// TIA Portal project "Multi_PLC_OPC_UA_Project" (V17)

(* hardware
DEVICE "S7-1200 station_1"  S7-1200 Station
   slot 0: "Rack_0"  S7-1200 Rack  Rack  V1.0
   slot 1: "PLC1_Loading"  CPU 1214C DC/DC/DC  6ES7 214-1AG40-0XB0  V4.5
DEVICE "S7-1200 station_2"  S7-1200 Station
   slot 0: "Rack_0"  S7-1200 Rack  Rack  V1.0
   slot 1: "PLC2_Testing"  CPU 1214C DC/DC/DC  6ES7 214-1AG40-0XB0  V4.5
DEVICE "HMI_Main"  KTP700 Basic PN
   slot 0: "HMI_Main"  KTP700 Basic PN  6AV2 123-2GB03-0AX0  17.0.0.0
   slot 1: "HMI_RT_1"  KTP700 Basic PN  6AV2 123-2GB03-0AX0  17.0.0.0
   slot 5: "HMI_Main.IE_CP_1"  PROFINET Interface  17.0.0.0
      slot 1: "PROFINET Interface_1"  PROFINET Interface
         slot 1: "Port_1"  Port
*)

// ===== PLC "PLC1_Loading"  CPU 1214C DC/DC/DC =====

VAR_GLOBAL   // PLC tag table "Default tag table"
   "PB_Start_Physical" AT %I0.0 : Bool;
   "PB_Stop_Physical" AT %I0.1 : Bool;
   "Conveyor_Run" AT %Q0.0 : Bool;
   "Light_Green" AT %Q0.1 : Bool;
   "Part_Sensor" AT %I0.2 : Bool;
   "Clock_Byte" AT %MB10 : Byte;
   "Clock_10Hz" AT %M10.0 : Bool;
   "Clock_5Hz" AT %M10.1 : Bool;
   "Clock_2.5Hz" AT %M10.2 : Bool;
   "Clock_2Hz" AT %M10.3 : Bool;
   "Clock_1.25Hz" AT %M10.4 : Bool;
   "Clock_1Hz" AT %M10.5 : Bool;
   "Clock_0.625Hz" AT %M10.6 : Bool;
   "Clock_0.5Hz" AT %M10.7 : Bool;
END_VAR

DATA_BLOCK "DB_PLC1_Commands"   // DB1
{ S7_Optimized_Access := 'FALSE' }
VERSION : 0.1
   VAR
      PB_Start : Bool;
      PB_Stop : Bool;
   END_VAR
BEGIN
END_DATA_BLOCK

DATA_BLOCK "DB_PLC1_Status"   // DB2
{ S7_Optimized_Access := 'FALSE' }
VERSION : 0.1
   VAR
      Conveyor_Run : Bool;
      Part_Sensor : Bool;
      Light_Green : Bool;
      Machine_Status : Int;
   END_VAR
BEGIN
END_DATA_BLOCK

DATA_BLOCK "DB_PLC1_To_PLC2"   // DB3
{ S7_Optimized_Access := 'FALSE' }
VERSION : 0.1
   VAR
      Part_Ready : Bool;
   END_VAR
BEGIN
END_DATA_BLOCK

DATA_BLOCK "DB_From_PLC2"   // DB6
{ S7_Optimized_Access := 'FALSE' }
VERSION : 0.1
   VAR
      Part_Done : Bool;
   END_VAR
BEGIN
END_DATA_BLOCK

ORGANIZATION_BLOCK "Main"   // OB1, LAD, ProgramCycle
TITLE = "Main Program Sweep (Cycle)"
{ S7_Optimized_Access := 'TRUE' }
VERSION : 0.1
   VAR_INPUT
      Initial_Call : Bool;   // Initial call of this OB
      Remanence : Bool;   // =True, if remanent data are available
   END_VAR
BEGIN

REGION Network 1
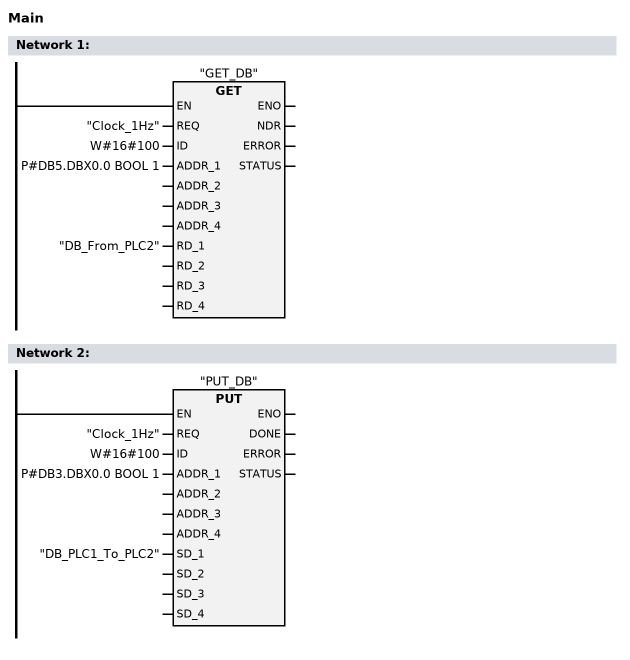
   "GET_DB"(REQ := "Clock_1Hz", ID := W#16#100, ADDR_1 := P#DB5.DBX0.0 BOOL 1, RD_1 := "DB_From_PLC2");   // GET
END_REGION

REGION Network 2
   "PUT_DB"(REQ := "Clock_1Hz", ID := W#16#100, ADDR_1 := P#DB3.DBX0.0 BOOL 1, SD_1 := "DB_PLC1_To_PLC2");   // PUT
END_REGION

REGION Network 3 (SCL)
   "DB_PLC1_Commands".PB_Start := "PB_Start_Physical";
   "DB_PLC1_Commands".PB_Stop := "PB_Stop_Physical";

   "Part_Sensor" := "DB_PLC1_Status".Part_Sensor;

   IF "DB_PLC1_Commands".PB_Start THEN

       "DB_PLC1_Status".Conveyor_Run := TRUE;
       "DB_PLC1_Status".Light_Green := TRUE;
       "DB_PLC1_Status".Machine_Status := 1;

   END_IF;

   IF "DB_PLC1_Commands".PB_Stop THEN

       "DB_PLC1_Status".Conveyor_Run := FALSE;
       "DB_PLC1_Status".Light_Green := FALSE;

       "DB_PLC1_To_PLC2".Part_Ready := FALSE;

       "DB_PLC1_Status".Machine_Status := 0;

   END_IF;


   IF "DB_PLC1_Status".Part_Sensor  AND NOT "DB_PLC1_To_PLC2".Part_Ready THEN

       "DB_PLC1_Status".Conveyor_Run := FALSE;

       "DB_PLC1_To_PLC2".Part_Ready := TRUE;

   END_IF;

   IF "DB_PLC1_To_PLC2".Part_Ready THEN

       "DB_PLC1_Status".Conveyor_Run := FALSE;

   END_IF;


   IF "DB_From_PLC2".Part_Done THEN


       "DB_PLC1_To_PLC2".Part_Ready := FALSE;

   END_IF;


   IF NOT "DB_PLC1_To_PLC2".Part_Ready
       AND "DB_PLC1_Commands".PB_Start THEN

       "DB_PLC1_Status".Conveyor_Run := TRUE;

   END_IF;


   "Conveyor_Run" := "DB_PLC1_Status".Conveyor_Run;

   "Light_Green" := "DB_PLC1_Status".Light_Green;
END_REGION
END_ORGANIZATION_BLOCK

// ===== PLC "PLC2_Testing"  CPU 1214C DC/DC/DC =====

VAR_GLOBAL   // PLC tag table "Default tag table"
   "PB_Start_Physical" AT %I0.0 : Bool;
   "PB_Stop_Physical" AT %I0.1 : Bool;
   "Conveyor_Run" AT %Q0.0 : Bool;
   "Light_Red" AT %Q0.1 : Bool;
   "Clock_Byte" AT %MB10 : Byte;
   "Clock_10Hz" AT %M10.0 : Bool;
   "Clock_5Hz" AT %M10.1 : Bool;
   "Clock_2.5Hz" AT %M10.2 : Bool;
   "Clock_2Hz" AT %M10.3 : Bool;
   "Clock_1.25Hz" AT %M10.4 : Bool;
   "Clock_1Hz" AT %M10.5 : Bool;
   "Clock_0.625Hz" AT %M10.6 : Bool;
   "Clock_0.5Hz" AT %M10.7 : Bool;
END_VAR

DATA_BLOCK "DB_PLC2_Commands"   // DB1
{ S7_Optimized_Access := 'FALSE' }
VERSION : 0.1
   VAR
      PB_Start : Bool;
      PB_Stop : Bool;
   END_VAR
BEGIN
END_DATA_BLOCK

DATA_BLOCK "DB_PLC2_Status"   // DB2
{ S7_Optimized_Access := 'FALSE' }
VERSION : 0.1
   VAR
      Conveyor_Run : Bool;
      Part_Ready_Old : Bool;
      Light_Red : Bool;
      Part_Count_Tested : Int;
      Quality_Pass : Bool;
      Machine_Status : Int;
   END_VAR
BEGIN
END_DATA_BLOCK

DATA_BLOCK "DB_From_PLC1"   // DB3
{ S7_Optimized_Access := 'FALSE' }
VERSION : 0.1
   VAR
      Part_Ready : Bool;
   END_VAR
BEGIN
END_DATA_BLOCK

DATA_BLOCK "DB_PLC2_To_PLC1"   // DB5
{ S7_Optimized_Access := 'FALSE' }
VERSION : 0.1
   VAR
      Part_Done : Bool;
   END_VAR
BEGIN
END_DATA_BLOCK

DATA_BLOCK "testing_sequence_DB"   // DB7
{ S7_Optimized_Access := 'TRUE' }
VERSION : 0.1
// stored: InstanceOfName testing_sequence
"testing_sequence"
BEGIN
END_DATA_BLOCK

FUNCTION_BLOCK "testing_sequence"   // FB1, SCL
{ S7_Optimized_Access := 'TRUE' }
VERSION : 0.1
   VAR
      "Step" : Int;
      Process_Timer : TON_TIME;
   END_VAR
BEGIN
   "DB_PLC2_Commands".PB_Start := "PB_Start_Physical";
   "DB_PLC2_Commands".PB_Stop := "PB_Stop_Physical";


   IF "DB_PLC2_Commands".PB_Start THEN

       "DB_PLC2_Status".Conveyor_Run := TRUE;
       "DB_PLC2_Status".Light_Red := TRUE;
       "DB_PLC2_Status".Machine_Status := 1;

   END_IF;


   IF "DB_PLC2_Commands".PB_Stop THEN

       "DB_PLC2_Status".Conveyor_Run := FALSE;
       "DB_PLC2_Status".Light_Red := FALSE;
       "DB_PLC2_Status".Machine_Status := 0;

       #Step := 0;

       #Process_Timer(
                      IN := FALSE,
                      PT := T#2s
       );

       "DB_PLC2_To_PLC1".Part_Done := FALSE;

   END_IF;


   CASE #Step OF

       0:
           #Process_Timer(
                          IN := FALSE,
                          PT := T#2s
           );

           "DB_PLC2_To_PLC1".Part_Done := FALSE;


           IF "DB_From_PLC1".Part_Ready THEN
               "DB_PLC2_Status".Part_Count_Tested :=
               "DB_PLC2_Status".Part_Count_Tested + 1;

               #Step := 10;

           END_IF;

       10:

           #Process_Timer(
                          IN := TRUE,
                          PT := T#2s
           );

           IF #Process_Timer.Q THEN
               #Step := 20;

           END_IF;

       20:
           #Process_Timer(
                          IN := FALSE,
                          PT := T#2s
           );

           "DB_PLC2_To_PLC1".Part_Done := TRUE;

           #Step := 30;

       30:
           IF NOT "DB_From_PLC1".Part_Ready THEN

               "DB_PLC2_To_PLC1".Part_Done := FALSE;

               #Step := 0;

           END_IF;

       ELSE

           #Step := 0;

           #Process_Timer(
                          IN := FALSE,
                          PT := T#2s
           );

           "DB_PLC2_To_PLC1".Part_Done := FALSE;

   END_CASE;
END_FUNCTION_BLOCK

ORGANIZATION_BLOCK "Main"   // OB1, LAD, ProgramCycle
TITLE = "Main Program Sweep (Cycle)"
{ S7_Optimized_Access := 'TRUE' }
VERSION : 0.1
   VAR_INPUT
      Initial_Call : Bool;   // Initial call of this OB
      Remanence : Bool;   // =True, if remanent data are available
   END_VAR
BEGIN

REGION Network 1
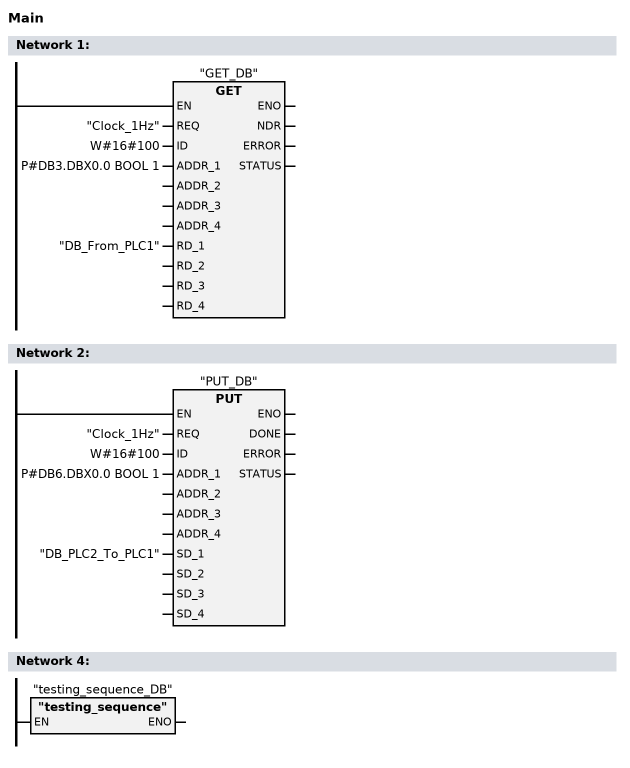
   "GET_DB"(REQ := "Clock_1Hz", ID := W#16#100, ADDR_1 := P#DB3.DBX0.0 BOOL 1, RD_1 := "DB_From_PLC1");   // GET
END_REGION

REGION Network 2
   "PUT_DB"(REQ := "Clock_1Hz", ID := W#16#100, ADDR_1 := P#DB6.DBX0.0 BOOL 1, SD_1 := "DB_PLC2_To_PLC1");   // PUT
END_REGION

REGION Network 3 (SCL)
   IF "GET_DB".ERROR THEN
       "DB_PLC2_Status".Machine_Status := 2;
   END_IF;
END_REGION

REGION Network 4
   RUNG wire#powerrail
      "testing_sequence_DB"()
   END_RUNG
   // the same network as SCL:
   "testing_sequence_DB"();   // "testing_sequence"
END_REGION
END_ORGANIZATION_BLOCK

(* ===== HMI "HMI_RT_1" =====
system functions are stored by id; their names below are inferred from use
connection "HMI_Connection_1": ETHERNET, SMART_S7_1200_OMS
connection "HMI_Connection_2": ETHERNET, SMART_S7_1200_OMS

HMI tags "Default tag table"
   "Tag_ScreenNumber" : UInt, internal
   "DB_PLC1_Commands_PB_Start" : Bool = PLC DB_PLC1_Commands.PB_Start AT %DB1.DBX0.0, 1 s
   "DB_PLC1_Commands_PB_Stop" : Bool = PLC DB_PLC1_Commands.PB_Stop AT %DB1.DBX0.1, 1 s
   "DB_PLC1_Status_Part_Count" : Int = PLC DB_PLC1_Status.Part_Count AT %DB2.DBW2, 1 s
   "DB_PLC2_Commands_PB_Start" : Bool = PLC DB_PLC2_Commands.PB_Start AT %DB1.DBX0.0, 1 s
   "DB_PLC2_Commands_PB_Stop" : Bool = PLC DB_PLC2_Commands.PB_Stop AT %DB1.DBX0.1, 1 s
   "DB_PLC2_Status_Part_Count_Tested" : Int = PLC DB_PLC2_Status.Part_Count_Tested AT %DB2.DBW2, 1 s
   "DB_From_PLC2_Part_Done" : Bool = PLC DB_From_PLC2.Part_Done AT %DB6.DBX0.0, 1 s
   "DB_PLC1_To_PLC2_Part_Ready" : Bool = PLC DB_PLC1_To_PLC2.Part_Ready AT %DB3.DBX0.0, 1 s
   "DB_PLC1_Status_Part_Count_not_tested" : Int = PLC DB_PLC1_Status.Part_Count AT %DB2.DBW2, 1 s
   "DB_PLC1_Status_Part_Sensor" : Bool = PLC DB_PLC1_Status.Part_Sensor AT %DB2.DBX0.1, 1 s
   "DB_PLC1_Status_Conveyor_Run" : Bool = PLC DB_PLC1_Status.Conveyor_Run AT %DB2.DBX0.0, 1 s
   "DB_PLC2_Status_Conveyor_Run" : Bool = PLC DB_PLC2_Status.Conveyor_Run AT %DB2.DBX0.0, 1 s
   "DB_From_PLC1_Part_Ready" : Bool = PLC DB_From_PLC1.Part_Ready AT %DB3.DBX0.0, 1 s

Template "Template_1" 800x480
   Button "Exit" at 714,429 size 71x50; TextOff 'Exit'; PictureOff "ExitRuntime_KTP700_Basic_PN_TR"; PictureOn "ExitRuntime_KTP700_Basic_PN_TR"
      on Release: StopRuntime(0)
   Button "Template_Button" at 614,429 size 71x50; TextOff 'Text'
   Button "Template_Button_1" at 514,429 size 71x50; TextOff 'Text'
   Button "Template_Button_2" at 414,429 size 71x50; TextOff 'Text'
   Button "Template_Button_3" at 314,429 size 71x50; TextOff 'Text'
   Button "Template_Button_4" at 214,429 size 71x50; TextOff 'Text'
   Button "Alarms" at 114,429 size 71x50; TextOff 'Alarms'; PictureOff "AlarmDisplay_KTP700_Basic_PN_TR"; PictureOn "AlarmDisplay_KTP700_Basic_PN_TR"
      on Release: function_ef3f5d25("Alarm window_Unacknowledged", -1)
   Button "Start screen" at 14,429 size 71x50; TextOff 'Start screen'; PictureOff "NavigateHome_KTP700_Basic_PN_TR"; PictureOn "NavigateHome_KTP700_Basic_PN_TR"
      on Release: ActivateScreen("Root screen", 0)
   SymbolicIOField "Symbolic_IO_Field_Screen" at 93,9 size 600x33; TextOff '0'; TextOn '1'; TextList "TextList_ScreenNames"
      ProcessValue <- "Tag_ScreenNumber"
      on Change: ActivateScreenByNumber("Tag_ScreenNumber", 0)
   DateTimeField "HmiScreenItemData" at 695,25 size 105x25
   DateTimeField "HmiScreenItemData_1" at 695,0 size 105x25
   GraphicView "Logo" at 0,0 size 91x51; Picture "Logo of HMI_1"

screen "Root screen" 800x480
   on GenerateScreen: SetTag("Tag_ScreenNumber", 1)
   TextField "HmiScreenItemData" at 63,10 size 640x25; Text 'Welcome to HMI_1 (KTP700 Basic+ PN)!'
   Button "Button_1" at 404,334 size 128x38; TextOff 'PLC1 START'
      on Press: SetBit("DB_PLC1_Commands_PB_Start")
      on Release: ResetBit("DB_PLC1_Commands_PB_Start")
   Button "Button_2" at 610,338 size 128x38; TextOff 'PLC1 STOP'
      on Release: ResetBit("DB_PLC1_Commands_PB_Stop")
      on Press: SetBit("DB_PLC1_Commands_PB_Stop")
   Button "Button_3" at 2,336 size 128x38; TextOff 'PLC2 START'
      on Release: ResetBit("DB_PLC2_Commands_PB_Start")
      on Press: SetBit("DB_PLC2_Commands_PB_Start")
   Button "Button_4" at 184,334 size 128x38; TextOff 'PLC2 STOP'
      on Release: ResetBit("DB_PLC2_Commands_PB_Stop")
      on Press: SetBit("DB_PLC2_Commands_PB_Stop")
   IOField "I/O field_1" at 168,396 size 96x32; FormatPattern 99999
      ProcessValue <- "DB_PLC2_Status_Part_Count_Tested"
   TextField "Text field_1" at 0,408 size 130x23; Text 'PARTS TESTED'
   Circle "Circle_1" at 402,79 size 60x60
      Appearance <- "DB_PLC1_To_PLC2_Part_Ready"
   Circle "Circle_2" at 22,79 size 60x60
      Appearance <- "DB_From_PLC2_Part_Done"
   TextField "Text field_2" at 389,146 size 113x23; Text 'PART READY'
   TextField "Text field_3" at 11,144 size 194x23; Text 'PART PROCESS FINISH'
   TextField "Text field_4" at 465,48 size 223x23; Text 'PLC 1 : LOADING STATION'
   TextField "Text field_5" at 89,43 size 223x23; Text 'PLC 2 : PROCESS STATION'
   TextField "Text field_6" at 543,89 size 118x23; Text 'Conveyor belt'
   TextField "Text field_8" at 513,187 size 122x23; Text 'SENSOR PART'
   Switch "Switch_1" at 648,185 size 64x32; CaptionText 'Switch'; TextOff 'OFF'; TextOn 'ON'
      ProcessValue <- "DB_PLC1_Status_Part_Sensor"
   TextField "Text field_11" at 9,254 size 216x23; Text 'PART READY FROM PLC 1'
   Circle "Circle_7" at 245,235 size 48x48
      Appearance <- "DB_From_PLC1_Part_Ready"
   TextField "Text field_12" at 401,254 size 210x23; Text 'PART DONE FROM PLC 2'
   Circle "Circle_8" at 625,241 size 48x48
      Appearance <- "DB_From_PLC2_Part_Done"
*)